FUNCTION_BLOCK WaterTank
  (* Standard: 61499-2 *)
  (* Version 0.1, 2015-00-10, syy, syy-PC *)
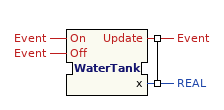
  EVENT_INPUT
    On;
    Off;
  END_EVENT
  EVENT_OUTPUT
    Update WITH x;
  END_EVENT
  VAR_OUTPUT
    x : REAL;
  END_VAR
  VAR
    C1x : REAL;
    k : REAL;
    d : REAL;
  END_VAR
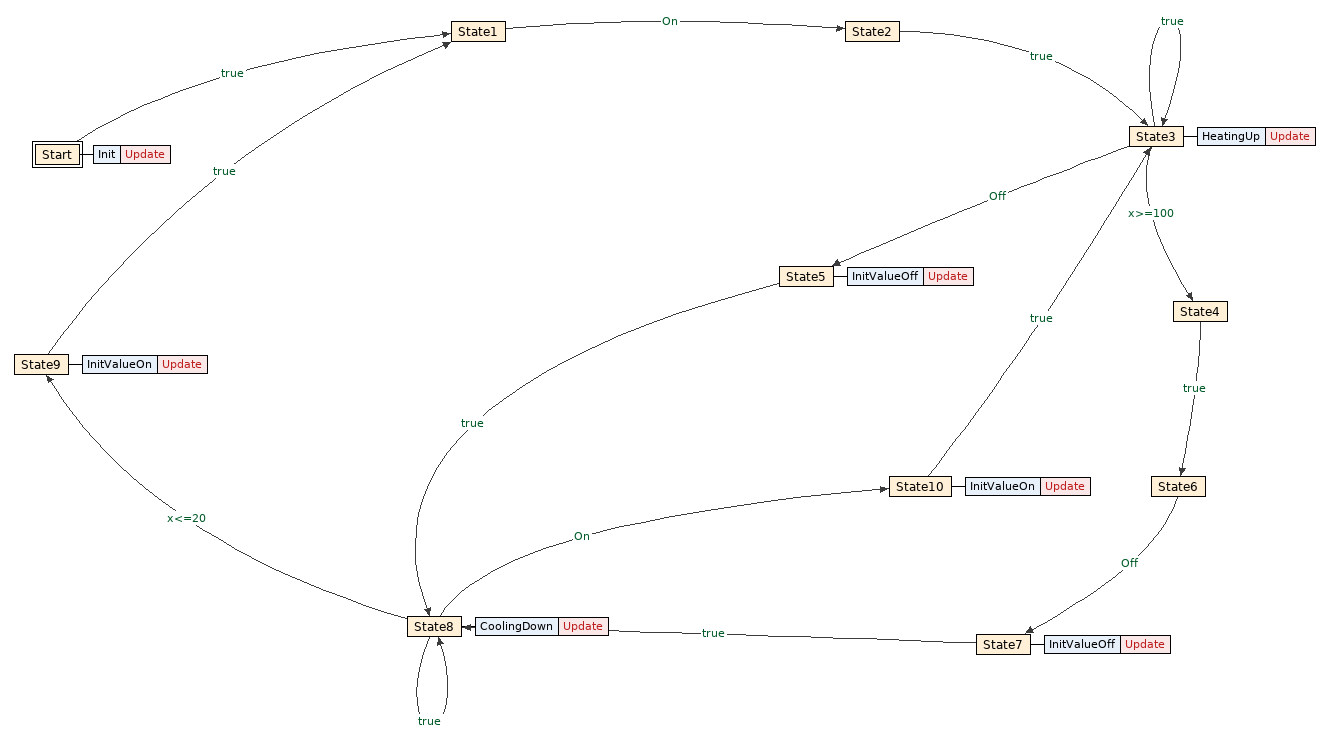
  EC_STATES
    Start : Init -> Update;
    State1;
    State2;
    State3 : HeatingUp -> Update;
    State4;
    State5 : InitValueOff -> Update;
    State6;
    State7 : InitValueOff -> Update;
    State8 : CoolingDown -> Update;
    State9 : InitValueOn -> Update;
    State10 : InitValueOn -> Update;
  END_STATES
  EC_TRANSITIONS
    Start TO State1 := true;
    State1 TO State2 := On;
    State2 TO State3 := true;
    State3 TO State4 := x>=100;
    State3 TO State5 := Off;
    State3 TO State3 := true;
    State4 TO State6 := true;
    State5 TO State8 := true;
    State6 TO State7 := Off;
    State7 TO State8 := true;
    State8 TO State9 := x<=20;
    State8 TO State10 := On;
    State8 TO State8 := true;
    State9 TO State1 := true;
    State10 TO State3 := true;
  END_TRANSITIONS
  ALGORITHM Init IN C:
me->x = 20;
me->C1x = -130;
me->d = 0.01;
me->k = 1;
printf("test\n");
  END_ALGORITHM
  ALGORITHM HeatingUp IN C:
me->x = (float) me->C1x*exp(-0.075*me->d*me->k) + 150.0;
me->k++;
printf("Temperature : %f\n", me->x);
  END_ALGORITHM
  ALGORITHM InitValueOff IN C:
me->k=0;
me->C1x=me->x;
  END_ALGORITHM
  ALGORITHM CoolingDown IN C:
me->x = (float) me->C1x*exp(-0.075*me->d*me->k);
me->k++;
//printf("Temperature : %f\n", me->x);
  END_ALGORITHM
  ALGORITHM InitValueOn IN C:
me->k=0;
me->C1x=me->x-150;
  END_ALGORITHM
END_FUNCTION_BLOCK
